Fanuc KAREL source: kb00177.KL

-- PROVISIONAL review KL for V940-1; original PC SHA256 6dc7dfab3c002505ab08600cc451cec1796ae841dec8d812c5da22749a067b68
-- Incomplete behavior may be omitted. Consult companion uncertainty JSON. Do not deploy.
PROGRAM KB00177
%NOLOCKGROUP
BEGIN
  -- V9_ZERO_TABLE_METADATA_HINT layout=0002_ascii; no indexed target words; source/name/runtime held
  -- UNRESOLVED_PC offsets 5-12; opcodes 9D,23
  -- UNRESOLVED_PC offsets 17-24; opcodes 9D,23
  -- UNRESOLVED_PC offsets 29-44; opcodes 2E,22,32,35
  -- UNRESOLVED_PC offsets 49-56; opcodes 9D,23
  -- UNRESOLVED_PC offsets 61-97; opcodes 27,22,22,22,1C,22,27,9D,31
  -- UNRESOLVED_PC offsets 102-106; opcodes 7F
END KB00177
